SUBAPPLICATION Abscheider (* Subapplication Type *)
  (* Standard: 61499-2 *)
  (* Version 1.0, 2023-01-29, Franz *)
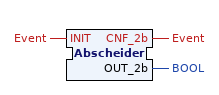
  EVENT_INPUT
    INIT; (* Service Initialization *)
  END_EVENT
  EVENT_OUTPUT
    CNF_2b; (* Execution Confirmation *)
  END_EVENT
  VAR_OUTPUT
    OUT_2b : BOOL;
  END_VAR
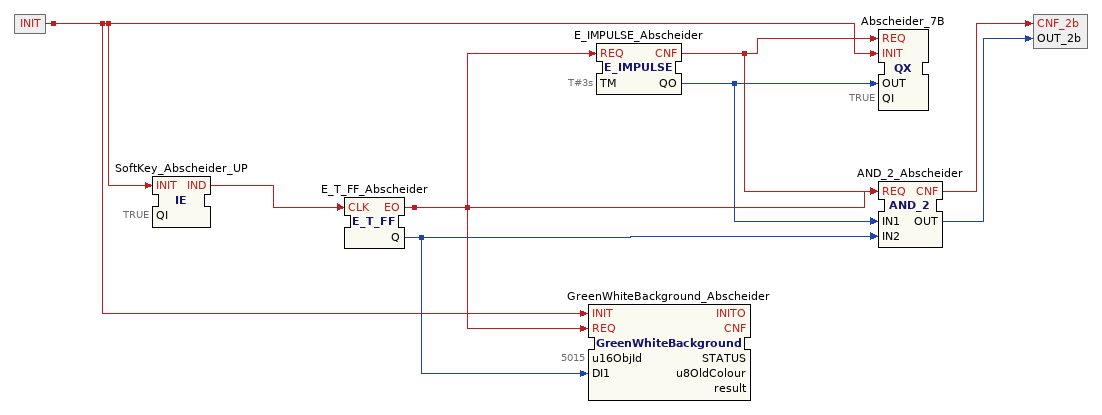
  FBS
    E_IMPULSE_Abscheider : E_IMPULSE(TM := T#3s);
    E_T_FF_Abscheider : E_T_FF;
    Abscheider_7B : QX(QI := TRUE);
    AND_2_Abscheider : AND_2;
    GreenWhiteBackground_Abscheider : GreenWhiteBackground(u16ObjId := 5015);
    SoftKey_Abscheider_UP : IE(QI := TRUE);
  END_FBS
  EVENT_CONNECTIONS
    E_T_FF_Abscheider.EO TO E_IMPULSE_Abscheider.REQ;
    E_IMPULSE_Abscheider.CNF TO AND_2_Abscheider.REQ;
    E_IMPULSE_Abscheider.CNF TO Abscheider_7B.REQ;
    E_T_FF_Abscheider.EO TO AND_2_Abscheider.REQ;
    E_T_FF_Abscheider.EO TO GreenWhiteBackground_Abscheider.REQ;
    AND_2_Abscheider.CNF TO CNF_2b;
    INIT TO GreenWhiteBackground_Abscheider.INIT;
    INIT TO Abscheider_7B.INIT;
    INIT TO SoftKey_Abscheider_UP.INIT;
    SoftKey_Abscheider_UP.IND TO E_T_FF_Abscheider.CLK;
  END_CONNECTIONS
  DATA_CONNECTIONS
    E_IMPULSE_Abscheider.QO TO AND_2_Abscheider.IN1;
    E_IMPULSE_Abscheider.QO TO Abscheider_7B.OUT;
    E_T_FF_Abscheider.Q TO AND_2_Abscheider.IN2;
    E_T_FF_Abscheider.Q TO GreenWhiteBackground_Abscheider.DI1;
    AND_2_Abscheider.OUT TO OUT_2b;
  END_CONNECTIONS
END_SUBAPPLICATION
